// TIA Portal project "metmoivc" (V15)

(* hardware
DEVICE "S7-1200 station_1"  S7-1200 Station
   slot 0: "Rack_0"  S7-1200 Rack  Rack  V1.0
   slot 1: "PLC_1"  CPU 1214C DC/DC/Rly  6ES7 214-1HG40-0XB0  V4.2
DEVICE "PC-System_1"  SIMATIC PC station
   slot 0: "SIMATIC PC station"  Rail  SIMATIC PC-Station  V1.0
      slot 125: "Stationmanager"  Station_Manager  V6.0.4
   slot 1: "HMI_RT_1"  WinCC RT Advanced  6AV2 104-0xxxx-xxxx  15.0.0.0
      slot 33792: "Host interface"  Host interface
   slot 2: "IE general_1"  IE General  IE_CP  V8.2.0
*)

// ===== PLC "PLC_1"  CPU 1214C DC/DC/Rly =====

VAR_GLOBAL   // PLC tag table "Default tag table"
   "Tag_1" AT %M50.0 : Bool;
   "Clock_Byte" AT %MB4 : Byte;
   "Clock_10Hz" AT %M4.0 : Bool;
   "Clock_5Hz" AT %M4.1 : Bool;
   "Clock_2.5Hz" AT %M4.2 : Bool;
   "Clock_2Hz" AT %M4.3 : Bool;
   "Clock_1.25Hz" AT %M4.4 : Bool;
   "Clock_1Hz" AT %M4.5 : Bool;
   "Clock_0.625Hz" AT %M4.6 : Bool;
   "Clock_0.5Hz" AT %M4.7 : Bool;
   "FirstScan" AT %M1.0 : Bool;
   "DiagStatusUpdate" AT %M1.1 : Bool;
   "AlwaysTRUE" AT %M1.2 : Bool;
   "AlwaysFALSE" AT %M1.3 : Bool;
   "Tag_2" AT %M50.1 : Bool;
   "Tag_3" AT %M50.2 : Bool;
   "Tag_4" AT %M50.3 : Bool;
   "Tag_5" AT %M50.4 : Bool;
   "Tag_6" AT %M50.5 : Bool;
   "Tag_7" AT %M50.6 : Bool;
   "Tag_8" AT %M50.7 : Bool;
   "Tag_9" AT %M51.0 : Bool;
   "Tag_10" AT %M51.1 : Bool;
   "TG1" AT %M51.2 : Bool;
   "TG2" AT %M51.3 : Bool;
   "TG3" AT %M51.4 : Bool;
   "TG4" AT %M51.5 : Bool;
   "TG5" AT %M51.6 : Bool;
   "TG6" AT %M51.7 : Bool;
   "TG7" AT %M52.0 : Bool;
END_VAR

VAR_GLOBAL   // PLC tag table "INPUT"
   "THERMOSTAT1" AT %M0.0 : Bool;
   "THERMOSTAT2" AT %M0.1 : Bool;
   "PROGRAM_SELECTOR3" AT %M0.2 : Bool;
   "PROGRAM_SELECTOR2" AT %M0.3 : Bool;
   "PROGRAM_SELECTOR1" AT %M0.4 : Bool;
   "TEMPERATURE1" AT %M0.5 : Bool;
   "TEMPERATURE2" AT %M0.6 : Bool;
   "START_BUTTON" AT %M0.7 : Bool;
   "LID_SWITCH" AT %M2.0 : Bool;
   "EMPTY_WATER" AT %M2.1 : Bool;
   "FULL_WATER" AT %M2.2 : Bool;
   "TG" AT %M2.3 : Bool;
   "Stop_all" AT %M2.4 : Bool;
   "Stop_count_start" AT %M2.5 : Bool;
END_VAR

VAR_GLOBAL   // PLC tag table "OUTPUT"
   "PROGRAM_STATUS3" AT %Q0.0 : Bool;
   "PROGRAM_STATUS2" AT %Q0.1 : Bool;
   "PROGRAM_STATUS1" AT %Q0.2 : Bool;
   "WATER_INLET_VALVE" AT %Q0.3 : Bool;
   "WATER_OUTLET_VALVE" AT %Q0.4 : Bool;
   "HEATING_ELEMENT" AT %Q0.5 : Bool;
   "MOTOR_FORWARD" AT %Q0.6 : Bool;
   "MOTOR_REVERSE" AT %Q0.7 : Bool;
   "PUMP" AT %Q1.0 : Bool;
END_VAR

VAR_GLOBAL   // PLC tag table "Tag_Present"
   "ET_Timer1" AT %MD10 : Time;
   "ET_Timer2" AT %MD14 : Time;
   "ET_Timer3" AT %MD18 : Time;
   "CV_Start" AT %MW22 : Int;
   "Water_Level" AT %MD26 : UDInt;
   "CV_Times_Stt2" AT %MW26 : Int;
   "Count_times_Stt2" AT %MW30 : Int;
   "Total_Time_Stt2" AT %MD100 : Time;
   "Total_time_stt3" AT %MD34 : Time;
   "ET_ton_stt2" AT %MD38 : Time;
   "ET_ton_stt3" AT %MD42 : Time;
   "ET_ton_stt2_1" AT %MD46 : Time;
END_VAR

VAR_GLOBAL   // PLC tag table "Tag_TG"
   "Lamp_Select1" AT %Q2.0 : Bool;
   "Lamp_Select2" AT %Q2.1 : Bool;
   "Lamp_Select3" AT %Q2.2 : Bool;
END_VAR

DATA_BLOCK "Data_block_1"   // DB12
{ S7_Optimized_Access := 'TRUE' }
VERSION : 0.1
   VAR
      ET_Time_1_stt2 : Time;
      ET_Time_2_stt2 : Time;
      ET_Time_1_stt4 : Time;
   END_VAR
BEGIN
END_DATA_BLOCK

// folder: System blocks/Program resources

DATA_BLOCK "IEC_Timer_0_DB"   // DB1
{ S7_Optimized_Access := 'TRUE' }
AUTHOR : Simatic
FAMILY : IEC
NAME : IEC_TMR
VERSION : 1.0
// stored: InstanceOfName IEC_TIMER
"IEC_TIMER"
BEGIN
END_DATA_BLOCK

DATA_BLOCK "IEC_Timer_0_DB_1"   // DB2
{ S7_Optimized_Access := 'TRUE' }
AUTHOR : Simatic
FAMILY : IEC
NAME : IEC_TMR
VERSION : 1.0
// stored: InstanceOfName IEC_TIMER
"IEC_TIMER"
BEGIN
END_DATA_BLOCK

DATA_BLOCK "IEC_Timer_0_DB_2"   // DB3
{ S7_Optimized_Access := 'TRUE' }
AUTHOR : Simatic
FAMILY : IEC
NAME : IEC_TMR
VERSION : 1.0
// stored: InstanceOfName IEC_TIMER
"IEC_TIMER"
BEGIN
END_DATA_BLOCK

DATA_BLOCK "Count_Simulation"   // DB4
{ S7_Optimized_Access := 'TRUE' }
AUTHOR : Simatic
FAMILY : IEC
NAME : UDCNTR
VERSION : 1.2
// stored: InstanceOfName IEC_UDCOUNTER
"IEC_UDCOUNTER"
BEGIN
END_DATA_BLOCK

DATA_BLOCK "count_empty"   // DB5
{ S7_Optimized_Access := 'TRUE' }
AUTHOR : Simatic
FAMILY : IEC
NAME : CNTR
VERSION : 1.0
// stored: InstanceOfName IEC_COUNTER
"IEC_COUNTER"
BEGIN
END_DATA_BLOCK

DATA_BLOCK "Count_Start"   // DB6
{ S7_Optimized_Access := 'TRUE' }
AUTHOR : Simatic
FAMILY : IEC
NAME : CNTR
VERSION : 1.0
// stored: InstanceOfName IEC_COUNTER
"IEC_COUNTER"
BEGIN
END_DATA_BLOCK

DATA_BLOCK "Count_Emty"   // DB7
{ S7_Optimized_Access := 'TRUE' }
AUTHOR : Simatic
FAMILY : IEC
NAME : CNTR
VERSION : 1.0
// stored: InstanceOfName IEC_COUNTER
"IEC_COUNTER"
BEGIN
END_DATA_BLOCK

DATA_BLOCK "Ton_Status2"   // DB8
{ S7_Optimized_Access := 'TRUE' }
AUTHOR : Simatic
FAMILY : IEC
NAME : IEC_TMR
VERSION : 1.0
// stored: InstanceOfName IEC_TIMER
"IEC_TIMER"
BEGIN
END_DATA_BLOCK

DATA_BLOCK "Ton_Status2_1"   // DB9
{ S7_Optimized_Access := 'TRUE' }
AUTHOR : Simatic
FAMILY : IEC
NAME : IEC_TMR
VERSION : 1.0
// stored: InstanceOfName IEC_TIMER
"IEC_TIMER"
BEGIN
END_DATA_BLOCK

DATA_BLOCK "Count_Full"   // DB10
{ S7_Optimized_Access := 'TRUE' }
AUTHOR : Simatic
FAMILY : IEC
NAME : CNTR
VERSION : 1.0
// stored: InstanceOfName IEC_COUNTER
"IEC_COUNTER"
BEGIN
END_DATA_BLOCK

DATA_BLOCK "Ton_Status3"   // DB11
{ S7_Optimized_Access := 'TRUE' }
AUTHOR : Simatic
FAMILY : IEC
NAME : IEC_TMR
VERSION : 1.0
// stored: InstanceOfName IEC_TIMER
"IEC_TIMER"
BEGIN
END_DATA_BLOCK

// folder: (top level)

FUNCTION "Status_1" : Void   // FC1, LAD
{ S7_Optimized_Access := 'TRUE' }
VERSION : 0.1
   VAR_TEMP   // added for the SCL form of the ladder/FBD networks
      _w1 : Bool;
   END_VAR
BEGIN

REGION Network 1: Status_1
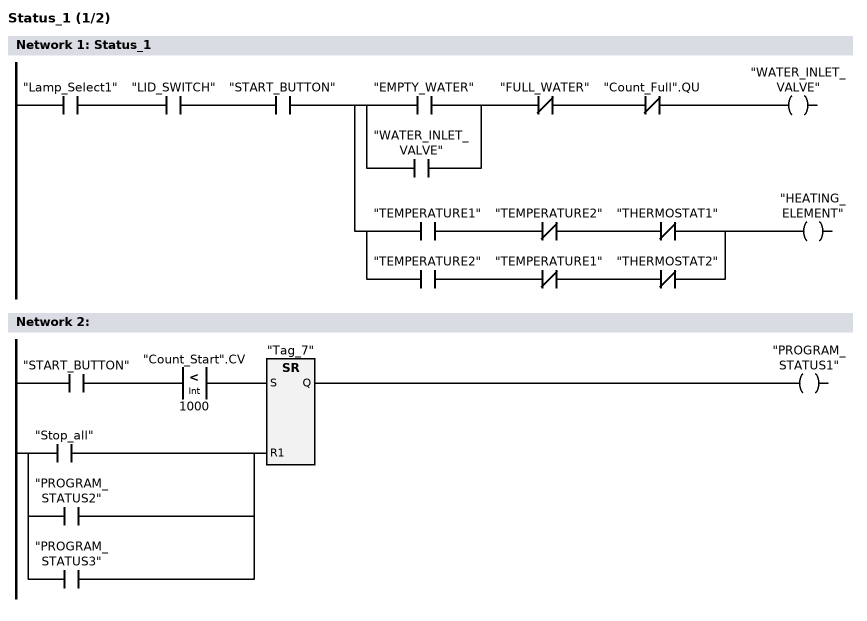
   RUNG wire#powerrail
      Contact( "Lamp_Select1" )
      Contact( "LID_SWITCH" )
      Contact( "START_BUTTON" )
      wire#w1
      Contact( "EMPTY_WATER" )
      wire#w2
      I_Contact( "FULL_WATER" )
      I_Contact( "Count_Full".QU )
      Coil( "WATER_INLET_VALVE" )
   END_RUNG
   RUNG wire#w1
      Contact( "WATER_INLET_VALVE" )
   END_RUNG wire#w2
   RUNG wire#w1
      Contact( "TEMPERATURE1" )
      I_Contact( "TEMPERATURE2" )
      I_Contact( "THERMOSTAT1" )
      wire#w3
      Coil( "HEATING_ELEMENT" )
   END_RUNG
   RUNG wire#w1
      Contact( "TEMPERATURE2" )
      I_Contact( "TEMPERATURE1" )
      I_Contact( "THERMOSTAT2" )
   END_RUNG wire#w3
   // the same network as SCL:
   #_w1 := "Lamp_Select1" AND "LID_SWITCH" AND "START_BUTTON";
   "WATER_INLET_VALVE" := #_w1 AND ("EMPTY_WATER" OR "WATER_INLET_VALVE") AND NOT "FULL_WATER" AND NOT "Count_Full".QU;
   "HEATING_ELEMENT" := #_w1 AND (("TEMPERATURE1" AND NOT "TEMPERATURE2" AND NOT "THERMOSTAT1") OR ("TEMPERATURE2" AND NOT "TEMPERATURE1" AND NOT "THERMOSTAT2"));
END_REGION

REGION Network 2
   RUNG wire#powerrail
      Contact( "START_BUTTON" )
      { S7_Templates := "SrcType := Int" } LT_Contact(in1 := "Count_Start".CV, in2 := 1000)
      S_SR(operand := "Tag_7", r1 := wire#w1)
      Coil( "PROGRAM_STATUS1" )
   END_RUNG
   RUNG wire#powerrail
      Contact( "Stop_all" )
   END_RUNG wire#w1
   RUNG wire#powerrail
      Contact( "PROGRAM_STATUS2" )
   END_RUNG wire#w1
   RUNG wire#powerrail
      Contact( "PROGRAM_STATUS3" )
   END_RUNG wire#w1
   // the same network as SCL:
   IF "START_BUTTON" AND ("Count_Start".CV < 1000) THEN
       "Tag_7" := TRUE;   // SR flip-flop
   END_IF;
   IF "Stop_all" OR "PROGRAM_STATUS2" OR "PROGRAM_STATUS3" THEN "Tag_7" := FALSE; END_IF;
   "PROGRAM_STATUS1" := "Tag_7";
END_REGION

REGION Network 3
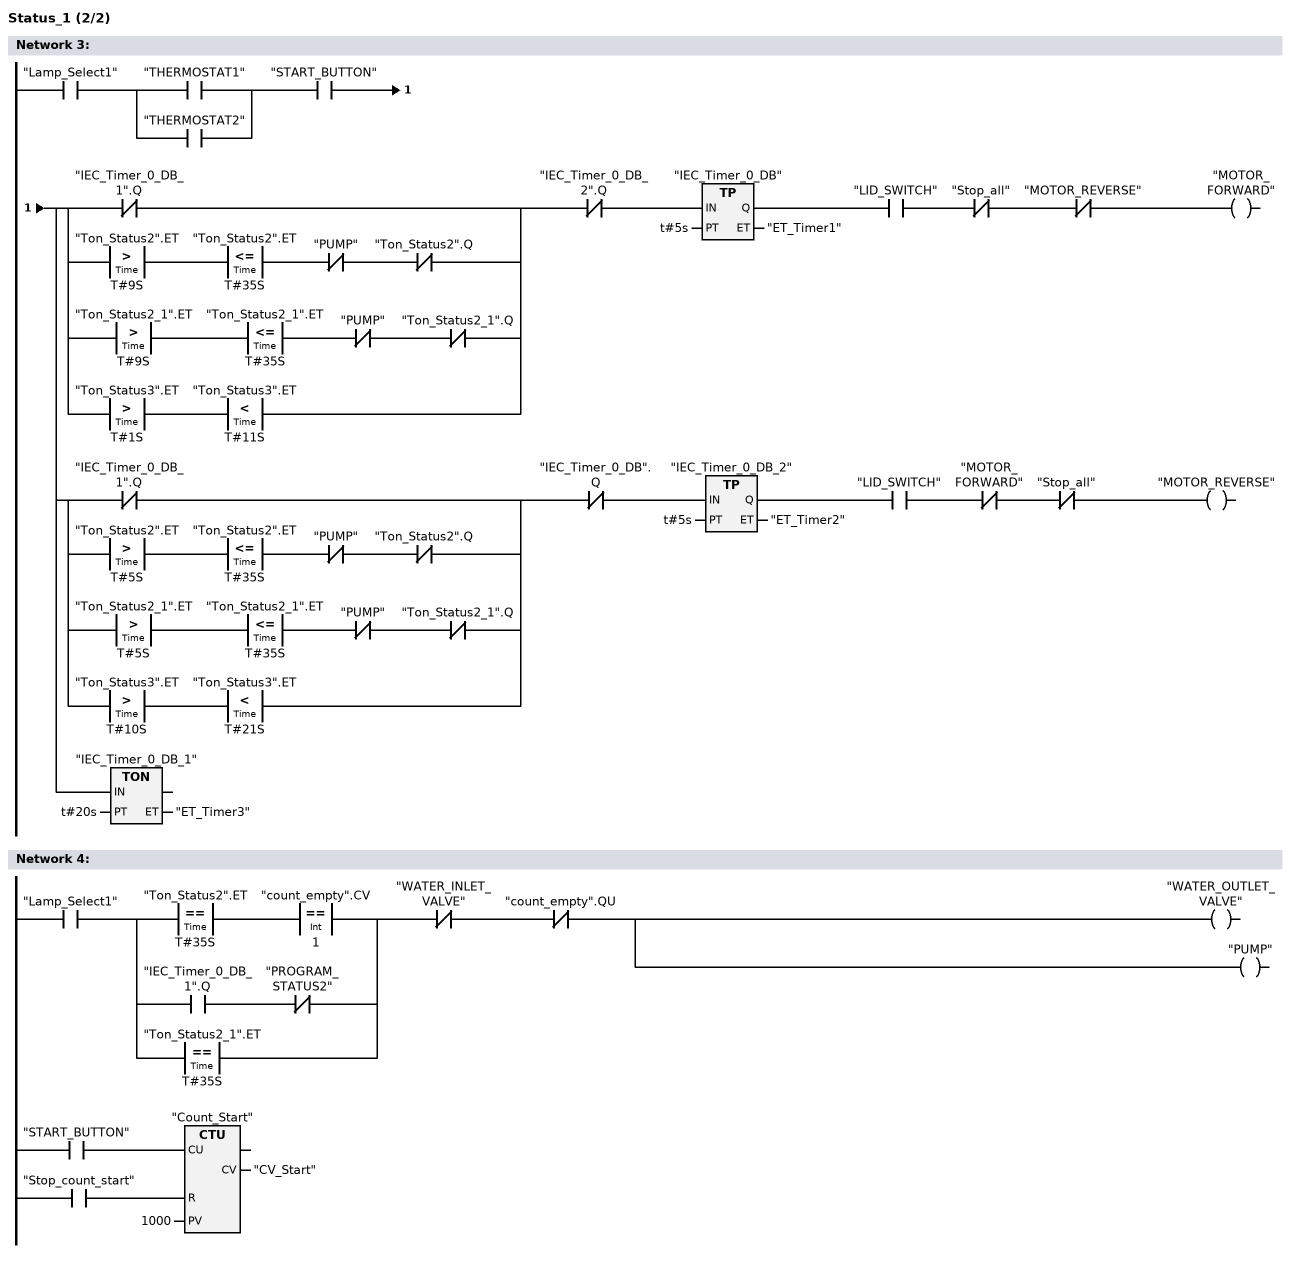
   #_w1 := "Lamp_Select1" AND ("THERMOSTAT1" OR "THERMOSTAT2") AND "START_BUTTON";
   "IEC_Timer_0_DB".TP(IN := #_w1 AND (NOT "IEC_Timer_0_DB_1".Q OR (("Ton_Status2".ET > T#9S) AND ("Ton_Status2".ET <= T#35S) AND NOT "PUMP" AND NOT "Ton_Status2".Q) OR (("Ton_Status2_1".ET > T#9S) AND ("Ton_Status2_1".ET <= T#35S) AND NOT "PUMP" AND NOT "Ton_Status2_1".Q) OR (("Ton_Status3".ET > T#1S) AND ("Ton_Status3".ET < T#11S))) AND NOT "IEC_Timer_0_DB_2".Q,
                       PT := t#5s,
                       ET => "ET_Timer1");
   "MOTOR_FORWARD" := "IEC_Timer_0_DB".Q AND "LID_SWITCH" AND NOT "Stop_all" AND NOT "MOTOR_REVERSE";
   "IEC_Timer_0_DB_2".TP(IN := #_w1 AND (NOT "IEC_Timer_0_DB_1".Q OR (("Ton_Status2".ET > T#5S) AND ("Ton_Status2".ET <= T#35S) AND NOT "PUMP" AND NOT "Ton_Status2".Q) OR (("Ton_Status2_1".ET > T#5S) AND ("Ton_Status2_1".ET <= T#35S) AND NOT "PUMP" AND NOT "Ton_Status2_1".Q) OR (("Ton_Status3".ET > T#10S) AND ("Ton_Status3".ET < T#21S))) AND NOT "IEC_Timer_0_DB".Q,
                         PT := t#5s,
                         ET => "ET_Timer2");
   "MOTOR_REVERSE" := "IEC_Timer_0_DB_2".Q AND "LID_SWITCH" AND NOT "MOTOR_FORWARD" AND NOT "Stop_all";
   "IEC_Timer_0_DB_1".TON(IN := #_w1, PT := t#20s, ET => "ET_Timer3");
END_REGION

REGION Network 4
   "WATER_OUTLET_VALVE" := "Lamp_Select1" AND ((("Ton_Status2".ET = T#35S) AND ("count_empty".CV = 1)) OR ("IEC_Timer_0_DB_1".Q AND NOT "PROGRAM_STATUS2") OR ("Ton_Status2_1".ET = T#35S)) AND NOT "WATER_INLET_VALVE" AND NOT "count_empty".QU;
   "PUMP" := "WATER_OUTLET_VALVE";
   "Count_Start".CTU(CU := "START_BUTTON", R := "Stop_count_start", PV := 1000, CV => "CV_Start");
END_REGION
END_FUNCTION

FUNCTION "Select_Program" : Void   // FC2, LAD
{ S7_Optimized_Access := 'TRUE' }
VERSION : 0.1
BEGIN

REGION Network 1
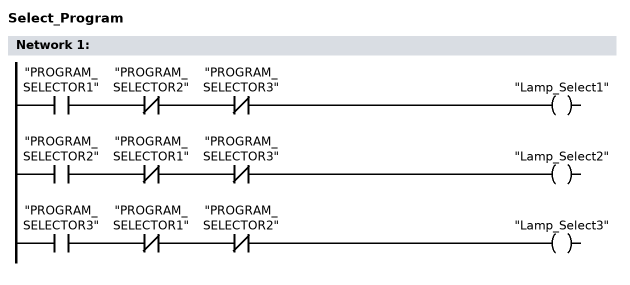
   RUNG wire#powerrail
      Contact( "PROGRAM_SELECTOR1" )
      I_Contact( "PROGRAM_SELECTOR2" )
      I_Contact( "PROGRAM_SELECTOR3" )
      Coil( "Lamp_Select1" )
   END_RUNG
   RUNG wire#powerrail
      Contact( "PROGRAM_SELECTOR2" )
      I_Contact( "PROGRAM_SELECTOR1" )
      I_Contact( "PROGRAM_SELECTOR3" )
      Coil( "Lamp_Select2" )
   END_RUNG
   RUNG wire#powerrail
      Contact( "PROGRAM_SELECTOR3" )
      I_Contact( "PROGRAM_SELECTOR1" )
      I_Contact( "PROGRAM_SELECTOR2" )
      Coil( "Lamp_Select3" )
   END_RUNG
   // the same network as SCL:
   "Lamp_Select1" := "PROGRAM_SELECTOR1" AND NOT "PROGRAM_SELECTOR2" AND NOT "PROGRAM_SELECTOR3";
   "Lamp_Select2" := "PROGRAM_SELECTOR2" AND NOT "PROGRAM_SELECTOR1" AND NOT "PROGRAM_SELECTOR3";
   "Lamp_Select3" := "PROGRAM_SELECTOR3" AND NOT "PROGRAM_SELECTOR1" AND NOT "PROGRAM_SELECTOR2";
END_REGION
END_FUNCTION

FUNCTION "Status_2" : Void   // FC3, LAD
{ S7_Optimized_Access := 'TRUE' }
VERSION : 0.1
   VAR_TEMP   // added for the SCL form of the ladder/FBD networks
      _w1 : Bool;
   END_VAR
BEGIN

REGION Network 1
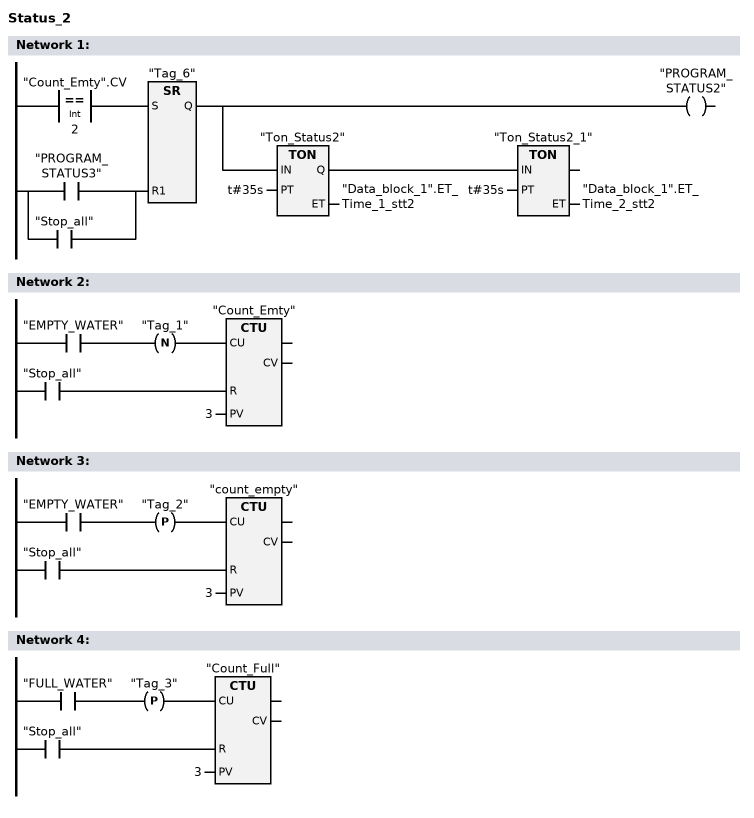
   IF "Count_Emty".CV = 2 THEN
       "Tag_6" := TRUE;   // SR flip-flop
   END_IF;
   IF "PROGRAM_STATUS3" OR "Stop_all" THEN "Tag_6" := FALSE; END_IF;
   "PROGRAM_STATUS2" := "Tag_6";
   "Ton_Status2".TON(IN := "Tag_6", PT := t#35s, ET => "Data_block_1".ET_Time_1_stt2);
   "Ton_Status2_1".TON(IN := "Ton_Status2".Q, PT := t#35s, ET => "Data_block_1".ET_Time_2_stt2);
END_REGION

REGION Network 2
   #_w1 := NOT "EMPTY_WATER" AND "Tag_1";   // falling edge
   "Tag_1" := "EMPTY_WATER";
   "Count_Emty".CTU(CU := #_w1, R := "Stop_all", PV := 3);
END_REGION

REGION Network 3
   #_w1 := "EMPTY_WATER" AND NOT "Tag_2";   // rising edge
   "Tag_2" := "EMPTY_WATER";
   "count_empty".CTU(CU := #_w1, R := "Stop_all", PV := 3);
END_REGION

REGION Network 4
   #_w1 := "FULL_WATER" AND NOT "Tag_3";   // rising edge
   "Tag_3" := "FULL_WATER";
   "Count_Full".CTU(CU := #_w1, R := "Stop_all", PV := 3);
END_REGION
END_FUNCTION

FUNCTION "Status_3" : Void   // FC4, LAD
{ S7_Optimized_Access := 'TRUE' }
VERSION : 0.1
BEGIN

REGION Network 1
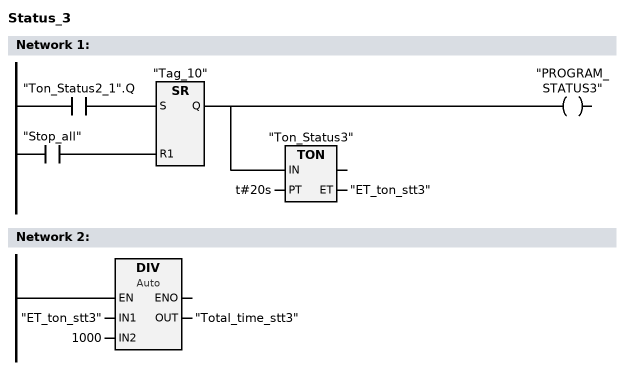
   IF "Ton_Status2_1".Q THEN
       "Tag_10" := TRUE;   // SR flip-flop
   END_IF;
   IF "Stop_all" THEN "Tag_10" := FALSE; END_IF;
   "PROGRAM_STATUS3" := "Tag_10";
   "Ton_Status3".TON(IN := "Tag_10", PT := t#20s, ET => "ET_ton_stt3");
END_REGION

REGION Network 2
   RUNG wire#powerrail
      Div(in1 := "ET_ton_stt3", in2 := 1000, out => "Total_time_stt3")
   END_RUNG
   // the same network as SCL:
   "Total_time_stt3" := "ET_ton_stt3" / 1000;
END_REGION
END_FUNCTION

FUNCTION "Simulation_Level_Water" : Void   // FC5, LAD
{ S7_Optimized_Access := 'TRUE' }
VERSION : 0.1
BEGIN

REGION Network 1
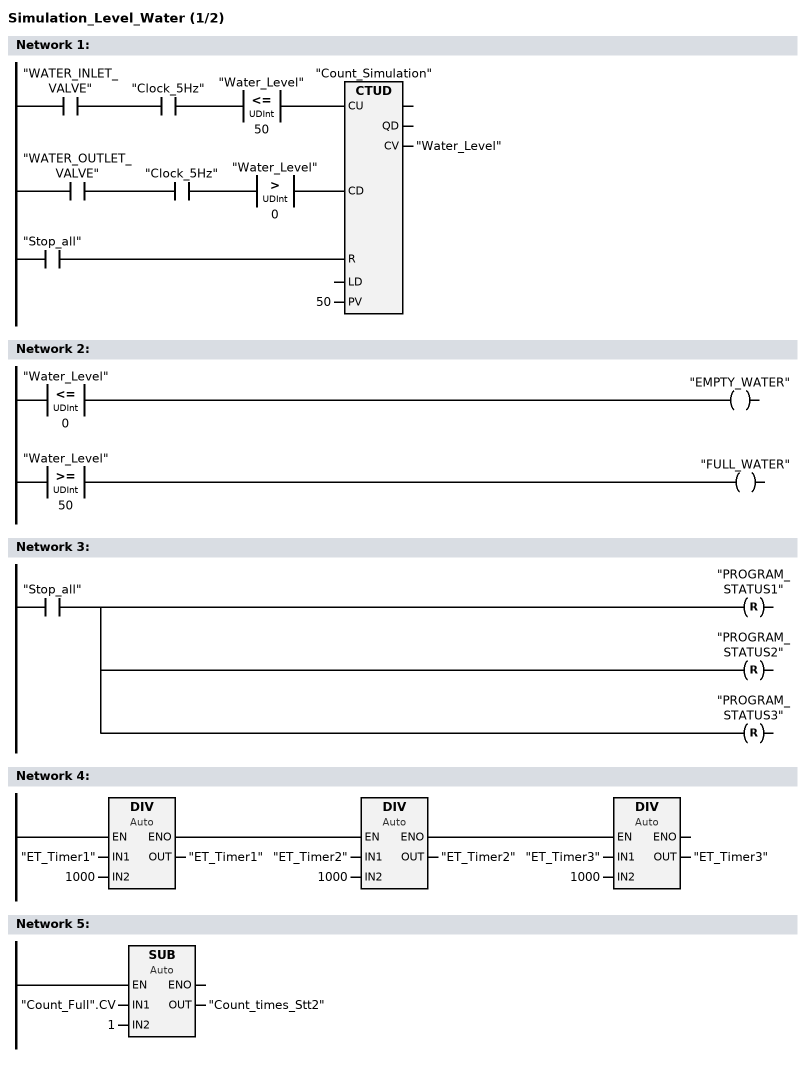
   "Count_Simulation".CTUD(CU := "WATER_INLET_VALVE" AND "Clock_5Hz" AND ("Water_Level" <= 50),
                           CD := "WATER_OUTLET_VALVE" AND "Clock_5Hz" AND ("Water_Level" > 0),
                           R := "Stop_all",
                           PV := 50,
                           CV => "Water_Level");
END_REGION

REGION Network 2
   RUNG wire#powerrail
      { S7_Templates := "SrcType := UDInt" } LE_Contact(in1 := "Water_Level", in2 := 0)
      Coil( "EMPTY_WATER" )
   END_RUNG
   RUNG wire#powerrail
      { S7_Templates := "SrcType := UDInt" } GE_Contact(in1 := "Water_Level", in2 := 50)
      Coil( "FULL_WATER" )
   END_RUNG
   // the same network as SCL:
   "EMPTY_WATER" := "Water_Level" <= 0;
   "FULL_WATER" := "Water_Level" >= 50;
END_REGION

REGION Network 3
   RUNG wire#powerrail
      Contact( "Stop_all" )
      wire#w1
      R_Coil( "PROGRAM_STATUS1" )
   END_RUNG
   RUNG wire#w1
      R_Coil( "PROGRAM_STATUS2" )
   END_RUNG
   RUNG wire#w1
      R_Coil( "PROGRAM_STATUS3" )
   END_RUNG
   // the same network as SCL:
   IF "Stop_all" THEN
       "PROGRAM_STATUS1" := FALSE;
       "PROGRAM_STATUS2" := FALSE;
       "PROGRAM_STATUS3" := FALSE;
   END_IF;
END_REGION

REGION Network 4
   RUNG wire#powerrail
      Div(in1 := "ET_Timer1", in2 := 1000, out => "ET_Timer1")
      Div(in1 := "ET_Timer2", in2 := 1000, out => "ET_Timer2")
      Div(in1 := "ET_Timer3", in2 := 1000, out => "ET_Timer3")
   END_RUNG
   // the same network as SCL:
   "ET_Timer1" := "ET_Timer1" / 1000;
   "ET_Timer2" := "ET_Timer2" / 1000;
   "ET_Timer3" := "ET_Timer3" / 1000;
END_REGION

REGION Network 5
   RUNG wire#powerrail
      Sub(in1 := "Count_Full".CV, in2 := 1, out => "Count_times_Stt2")
   END_RUNG
   // the same network as SCL:
   "Count_times_Stt2" := "Count_Full".CV - 1;
END_REGION

REGION Network 6
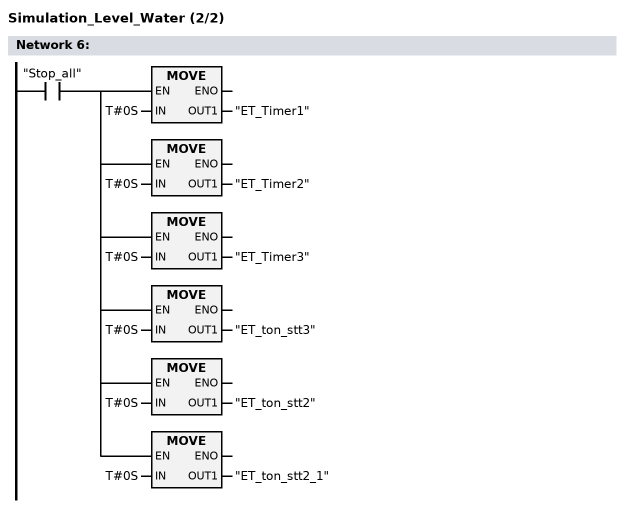
   RUNG wire#powerrail
      Contact( "Stop_all" )
      wire#w1
      Move(in := T#0S, out1 => "ET_Timer1")
   END_RUNG
   RUNG wire#w1
      Move(in := T#0S, out1 => "ET_Timer2")
   END_RUNG
   RUNG wire#w1
      Move(in := T#0S, out1 => "ET_Timer3")
   END_RUNG
   RUNG wire#w1
      Move(in := T#0S, out1 => "ET_ton_stt3")
   END_RUNG
   RUNG wire#w1
      Move(in := T#0S, out1 => "ET_ton_stt2")
   END_RUNG
   RUNG wire#w1
      Move(in := T#0S, out1 => "ET_ton_stt2_1")
   END_RUNG
   // the same network as SCL:
   IF "Stop_all" THEN
       "ET_Timer1" := T#0S;
       "ET_Timer2" := T#0S;
       "ET_Timer3" := T#0S;
       "ET_ton_stt3" := T#0S;
       "ET_ton_stt2" := T#0S;
       "ET_ton_stt2_1" := T#0S;
   END_IF;
END_REGION
END_FUNCTION

ORGANIZATION_BLOCK "Main"   // OB1, LAD, ProgramCycle
TITLE = "Main Program Sweep (Cycle)"
{ S7_Optimized_Access := 'TRUE' }
VERSION : 0.1
   VAR_INPUT
      Initial_Call : Bool;   // Initial call of this OB
      Remanence : Bool;   // =True, if remanent data are available
   END_VAR
   VAR_TEMP   // added for the SCL form of the ladder/FBD networks
      _w1 : Bool;
      _w2 : Bool;
      _w3 : Bool;
      _w4 : Bool;
   END_VAR
BEGIN

REGION Network 1
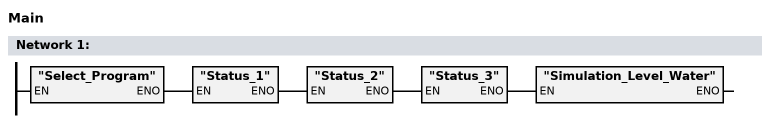
   RUNG wire#powerrail
      "Select_Program"()
      "Status_1"()
      "Status_2"()
      "Status_3"()
      "Simulation_Level_Water"()
   END_RUNG
   // the same network as SCL:
   "Select_Program"(ENO => #_w1);
   "Status_1"(EN := #_w1, ENO => #_w2);
   "Status_2"(EN := #_w2, ENO => #_w3);
   "Status_3"(EN := #_w3, ENO => #_w4);
   IF #_w4 THEN "Simulation_Level_Water"(); END_IF;
END_REGION
END_ORGANIZATION_BLOCK

(* ===== HMI "HMI_RT_1" =====
system functions are stored by id; their names below are inferred from use
connection "HMI_Connection_1": ETHERNET, S7_1200_OMS

HMI tags "Default tag table"
   "ET_Timer1" : Time = PLC ET_Timer1 AT %MD10, 1 s
   "ET_Timer2" : Time = PLC ET_Timer2 AT %MD14, 1 s
   "ET_Timer3" : Time = PLC ET_Timer3 AT %MD18, 1 s
   "PROGRAM_SELECTOR1" : Bool = PLC PROGRAM_SELECTOR1 AT %M0.4, 1 s
   "PROGRAM_SELECTOR2" : Bool = PLC PROGRAM_SELECTOR2 AT %M0.3, 1 s
   "PROGRAM_STATUS1" : Bool = PLC PROGRAM_STATUS1 AT %Q0.2, 1 s
   "PROGRAM_STATUS2" : Bool = PLC PROGRAM_STATUS2 AT %Q0.1, 1 s
   "PROGRAM_STATUS3" : Bool = PLC PROGRAM_STATUS3 AT %Q0.0, 1 s
   "START_BUTTON" : Bool = PLC START_BUTTON AT %M0.7, 1 s
   "PROGRAM_SELECTOR3" : Bool = PLC PROGRAM_SELECTOR3 AT %M0.2, 1 s
   "MOTOR_FORWARD" : Bool = PLC MOTOR_FORWARD AT %Q0.6, 1 s
   "MOTOR_REVERSE" : Bool = PLC MOTOR_REVERSE AT %Q0.7, 1 s
   "CV_Start" : Int = PLC CV_Start AT %MW22, 1 s
   "FULL_WATER" : Bool = PLC FULL_WATER AT %M2.2, 1 s
   "Lamp_Select1" : Bool = PLC Lamp_Select1 AT %Q2.0, 1 s
   "Lamp_Select2" : Bool = PLC Lamp_Select2 AT %Q2.1, 1 s
   "Lamp_Select3" : Bool = PLC Lamp_Select3 AT %Q2.2, 1 s
   "WATER_INLET_VALVE" : Bool = PLC WATER_INLET_VALVE AT %Q0.3, 1 s
   "WATER_OUTLET_VALVE" : Bool = PLC WATER_OUTLET_VALVE AT %Q0.4, 1 s
   "TEMPERATURE1" : Bool = PLC TEMPERATURE1 AT %M0.5, 1 s
   "TEMPERATURE2" : Bool = PLC TEMPERATURE2 AT %M0.6, 1 s
   "LID_SWITCH" : Bool = PLC LID_SWITCH AT %M2.0, 1 s
   "Water_Level" : UDInt = PLC Water_Level AT %MD26, 1 s
   "Stop_all" : Bool = PLC Stop_all AT %M2.4, 1 s
   "EMPTY_WATER" : Bool = PLC EMPTY_WATER AT %M2.1, 1 s
   "CV_Times_Stt2" : Int = PLC CV_Times_Stt2 AT %MW26, 1 s
   "THERMOSTAT1" : Bool = PLC THERMOSTAT1 AT %M0.0, 1 s
   "THERMOSTAT2" : Bool = PLC THERMOSTAT2 AT %M0.1, 1 s
   "HEATING_ELEMENT" : Bool = PLC HEATING_ELEMENT AT %Q0.5, 1 s
   "Count_times_Stt2" : Int = PLC Count_times_Stt2 AT %MW30, 1 s
   "Stop_count_start" : Bool = PLC Stop_count_start AT %M2.5, 1 s
   "Total_Time_Stt2" : Time = PLC Total_Time_Stt2 AT %MD100, 1 s
   "Total_time_stt3" : Time = PLC Total_time_stt3 AT %MD34, 1 s

screen "Screen_1" 1920x1080
   SymbolLibrary "Symbol library_14" at 715,489 size 120x68
      Appearance <- "HEATING_ELEMENT"
   SymbolLibrary "Symbol library_7" at 451,381 size 58x51
      Appearance <- "WATER_INLET_VALVE"
   SymbolLibrary "Symbol library_5" at 469,631 size 31x40
      Appearance <- "WATER_OUTLET_VALVE"
   Switch "Switch_1" at 59,369 size 120x62; CaptionText 'Select_1'; TextOff 'OFF'; TextOn 'ON'
      on SwitchOn: SetBit("PROGRAM_SELECTOR1")
      on SwitchOff: ResetBit("PROGRAM_SELECTOR1")
      ProcessValue <- "PROGRAM_SELECTOR1"
   Circle "Circle_1" at 200,383 size 48x48
      Appearance <- "Lamp_Select1"
   TextField "Text field_1" at 430,373 size 15x22; Text 'Text'
   Switch "Switch_2" at 59,439 size 120x65; CaptionText 'Select_2'; TextOff 'OFF'; TextOn 'ON'
      on SwitchOn: SetBit("PROGRAM_SELECTOR2")
      on SwitchOff: ResetBit("PROGRAM_SELECTOR2")
   Switch "Switch_3" at 59,508 size 120x63; CaptionText 'Select_3'; TextOff 'OFF'; TextOn 'ON'
      on SwitchOn: SetBit("PROGRAM_SELECTOR3")
      on SwitchOff: ResetBit("PROGRAM_SELECTOR3")
   Switch "Switch_4" at 59,586 size 120x63; TextOn 'ON'; CaptionText 'Start'; TextOff 'OFF'
      on SwitchOn: SetBit("START_BUTTON")
      on SwitchOff: ResetBit("START_BUTTON")
   Circle "Circle_2" at 200,604 size 48x48
      Appearance <- "START_BUTTON"
   Circle "Circle_3" at 199,527 size 48x48
      Appearance <- "Lamp_Select3"
   Circle "Circle_4" at 199,458 size 48x48
      Appearance <- "Lamp_Select2"
   IOField "I/O field_1" at 187,668 size 65x30; FormatPattern 99999
      ProcessValue <- "CV_Start"
   TextField "Text field_2" at 58,668 size 118x22; Text 'COUNT_START'
   TextField "Text field_3" at 428,2 size 444x39; Text 'Washing Machine Automation'
   SymbolLibrary "Symbol library_2" at 579,646 size 47x65
      Appearance <- "MOTOR_FORWARD"
   SymbolLibrary "Symbol library_3" at 483,406 size 246x248
   SymbolLibrary "Symbol library_1" at 738,402 size 73x43
      Appearance <- "FULL_WATER"
   SymbolLibrary "Symbol library_4" at 739,617 size 73x43
      Appearance <- "EMPTY_WATER"
   TextField "Text field_4" at 732,373 size 93x22; Text 'Full_sensor'
      Appearance <- "FULL_WATER"
   TextField "Text field_5" at 732,667 size 111x22; Text 'Empty_sensor'
      Appearance <- "EMPTY_WATER"
   SymbolLibrary "Symbol library_6" at 466,667 size 28x65
      Appearance <- "WATER_OUTLET_VALVE"
   IOField "I/O field_2" at 190,256 size 47x37; FormatPattern 9
      ProcessValue <- "ET_Timer2"
   Circle "Circle_5" at 73,174 size 48x48
      Appearance <- "MOTOR_FORWARD"
   Circle "Circle_6" at 187,173 size 48x48
      Appearance <- "MOTOR_REVERSE"
   TextField "Text field_6" at 90,110 size 125x22; Text 'STATUS MOTOR'
   TextField "Text field_7" at 74,225 size 41x22; Text 'Time'
   TextField "Text field_8" at 65,150 size 70x20; Text 'FORWARD'
   TextField "Text field_9" at 182,150 size 61x20; Text 'RESERVE'
   IOField "I/O field_3" at 75,255 size 46x39; FormatPattern 9
      ProcessValue <- "ET_Timer1"
   TextField "Text field_10" at 187,223 size 41x22; Text 'Time'
   SymbolLibrary "Symbol library_9" at 614,751 size 42x39
      Appearance <- "WATER_OUTLET_VALVE"
   SymbolLibrary "Symbol library_10" at 515,737 size 101x62
      Appearance <- "WATER_OUTLET_VALVE"
   IOField "I/O field_4" at 529,172 size 53x38; FormatPattern 99
      ProcessValue <- "ET_Timer3"
   SymbolLibrary "Symbol library_11" at 468,730 size 50x44
      Appearance <- "WATER_OUTLET_VALVE"
   TextField "Text field_13" at 448,339 size 81x27; Text 'Valve in'
      Appearance <- "WATER_INLET_VALVE"
   SymbolLibrary "Symbol library_8" at 388,377 size 65x29
      Appearance <- "WATER_INLET_VALVE"
   TextField "Text field_14" at 527,805 size 65x29; Text 'Pump'
      Appearance <- "WATER_OUTLET_VALVE"
   TextField "Text field_15" at 430,654 size 27x98; Text 'Valve Out'
      Appearance <- "WATER_OUTLET_VALVE"
   SymbolLibrary "Symbol library_12" at 631,799 size 35x53
      Appearance <- "WATER_OUTLET_VALVE"
   SymbolLibrary "Symbol library_13" at 325,379 size 53x35
      Appearance <- "WATER_INLET_VALVE"
   DateTimeField "Date/time field_1" at 517,41 size 259x36
   Circle "Circle_7" at 530,95 size 49x49
      Appearance <- "PROGRAM_STATUS1"
   Switch "Switch_5" at 100,780 size 109x64; CaptionText 'Temp_Control'; TextOff '2'; TextOn '1'
      on SwitchOn: SetBit("TEMPERATURE1"); ResetBit("TEMPERATURE2")
      on SwitchOff: SetBit("TEMPERATURE2"); ResetBit("TEMPERATURE1")
   Switch "Switch_7" at 1057,132 size 118x65; TextOn 'ON'; CaptionText 'LID Switch'; TextOff 'OFF'
      on SwitchOff: ResetBit("LID_SWITCH")
      on SwitchOn: SetBit("LID_SWITCH")
      ProcessValue <- "LID_SWITCH"
   Bar "Bar_1" at 483,414 size 246x240; MinimumValue 0; MaximumValue 50
      ProcessValue <- "Water_Level"
   Button "Button_1" at 58,711 size 119x32; TextOff 'Reset System'
      on Press: SetBit("Stop_all")
      on Release: ResetBit("Stop_all")
   TextField "Text field_16" at 522,141 size 67x22; Text 'Status 1'
   Circle "Circle_8" at 613,95 size 49x49
      Appearance <- "PROGRAM_STATUS2"
   TextField "Text field_17" at 606,141 size 67x22; Text 'Status 2'
   Circle "Circle_9" at 696,95 size 49x49
      Appearance <- "PROGRAM_STATUS3"
   TextField "Text field_18" at 691,141 size 67x22; Text 'Status 3'
   TextField "Text field_19" at 535,214 size 41x22; Text 'Time'
   TextField "Text field_20" at 617,214 size 49x22; Text 'Times'
   IOField "I/O field_6" at 614,172 size 53x38; FormatPattern 9
      ProcessValue <- "Count_times_Stt2"
   Switch "Switch_6" at 1012,228 size 103x64; CaptionText 'THERMOSTAT1'; TextOff 'OFF'; TextOn 'ON'
      on SwitchOn: SetBit("THERMOSTAT1")
      on SwitchOff: ResetBit("THERMOSTAT1")
      ProcessValue <- "THERMOSTAT1"
   Switch "Switch_8" at 1138,228 size 96x63; CaptionText 'THERMOSTAT2'; TextOff 'OFF'; TextOn 'ON'
      on SwitchOn: SetBit("THERMOSTAT2")
      on SwitchOff: ResetBit("THERMOSTAT2")
      ProcessValue <- "THERMOSTAT2"
   Button "Button_2" at 194,711 size 53x32; TextOff 'Reset'
      on Release: ResetBit("Stop_count_start")
      on Press: SetBit("Stop_count_start")
   IOField "I/O field_7" at 698,171 size 53x38; FormatPattern 99
      ProcessValue <- "Total_time_stt3"
   TextField "Text field_21" at 699,214 size 41x22; Text 'Time'
   TextField "Text field_22" at 732,553 size 93x22; Text 'Heating'
      Appearance <- "HEATING_ELEMENT"
   TextField "Text field_23" at 48,751 size 204x27; Text 'Temperature Control'
   TextField "Text field_12" at 1063,101 size 105x22; Text 'SIMULATION'
*)